TYPE ST130_Recipe_t :
STRUCT
    diLoadMixture_ms : DINT; // waiting time until mixture is fully loaded
    xUseVerLeft      : BOOL; // Is the left vertical picker element is used
    xUseVerRight     : BOOL; // Is the right vertical picker element is used
END_STRUCT
END_TYPE

(* stored: Version 1.1.0.1, ProductVersion 3.1.4024.6
   DUT ST130_Recipe_t: Id {41300b22-4f55-48a2-963a-64b2e064b0f7} *)
